// TIA Portal project "Contadores" (V16)

(* hardware
DEVICE "S7-1200 station_1"  S7-1200 Station
   slot 0: "Rack_0"  S7-1200 Rack  Rack  V1.0
   slot 1: "PLC_1"  CPU 1214C AC/DC/Rly  6ES7 214-1BG40-0XB0  V4.4
*)

// ===== PLC "PLC_1"  CPU 1214C AC/DC/Rly =====

VAR_GLOBAL   // PLC tag table "Tabla de variables estándar"
   "Flancos" AT %I0.0 : Bool;
   "Reset" AT %I0.1 : Bool;
   "Contador" AT %MW100 : Int;
   "Relé" AT %Q0.0 : Bool;
   "FlancosDesc" AT %I0.2 : Bool;
   "ResetDesc" AT %I0.3 : Bool;
   "ContadorDesc" AT %MW101 : Int;
   "INT ASC" AT %I0.4 : Bool;
   "INT DESC" AT %I0.5 : Bool;
   "RESET TO 0" AT %I0.6 : Bool;
   "RESET TO 10" AT %I0.7 : Bool;
   "OUT CTU" AT %Q0.1 : Bool;
   "OUT CTD" AT %Q0.2 : Bool;
   "MEMORIA" AT %MD100 : DWord;
END_VAR

// folder: System blocks/Program resources

DATA_BLOCK "IEC_Counter_0_DB"   // DB1
{ S7_Optimized_Access := 'TRUE' }
AUTHOR : Simatic
FAMILY : IEC
NAME : CNTR
VERSION : 1.0
// stored: InstanceOfName IEC_COUNTER
"IEC_COUNTER"
BEGIN
END_DATA_BLOCK

DATA_BLOCK "IEC_Counter_0_DB_1"   // DB2
{ S7_Optimized_Access := 'TRUE' }
AUTHOR : Simatic
FAMILY : IEC
NAME : CNTR
VERSION : 1.0
// stored: InstanceOfName IEC_COUNTER
"IEC_COUNTER"
BEGIN
END_DATA_BLOCK

DATA_BLOCK "IEC_Counter_0_DB_2"   // DB3
{ S7_Optimized_Access := 'TRUE' }
AUTHOR : Simatic
FAMILY : IEC
NAME : CNTR
VERSION : 1.0
// stored: InstanceOfName IEC_COUNTER
"IEC_COUNTER"
BEGIN
END_DATA_BLOCK

// folder: (top level)

ORGANIZATION_BLOCK "Main"   // OB1, LAD, ProgramCycle
TITLE = "Main Program Sweep (Cycle)"
{ S7_Optimized_Access := 'TRUE' }
VERSION : 0.1
   VAR_INPUT
      Initial_Call : Bool;   // Initial call of this OB
      Remanence : Bool;   // =True, if remanent data are available
   END_VAR
BEGIN

REGION Network 1
   // Contador de flanco ascendente CTU
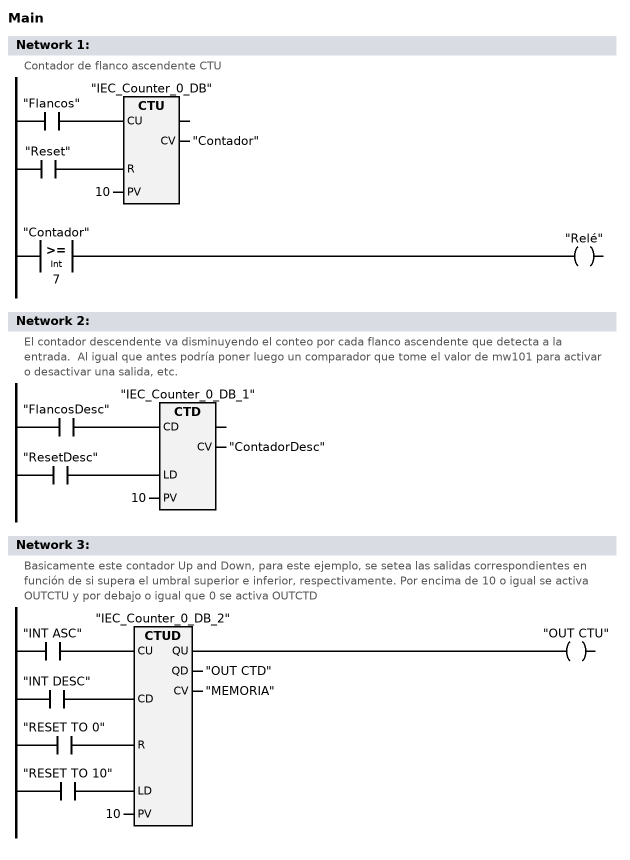
   "IEC_Counter_0_DB".CTU(CU := "Flancos", R := "Reset", PV := 10, CV => "Contador");
   "Relé" := "Contador" >= 7;
END_REGION

REGION Network 2
   // El contador descendente va disminuyendo el conteo por cada flanco ascendente que detecta a la entrada.  Al igual que antes podría poner luego un comparador que tome el valor de mw101 para activar o desactivar una salida, etc.
   "IEC_Counter_0_DB_1".CTD(CD := "FlancosDesc", LD := "ResetDesc", PV := 10, CV => "ContadorDesc");
END_REGION

REGION Network 3
   // Basicamente este contador Up and Down, para este ejemplo, se setea las salidas correspondientes en función de si supera el umbral superior e inferior, respectivamente. Por encima de 10 o igual se activa OUTCTU y por debajo o igual que 0 se activa OUTCTD
   "IEC_Counter_0_DB_2".CTUD(CU := "INT ASC",
                           CD := "INT DESC",
                           R := "RESET TO 0",
                           LD := "RESET TO 10",
                           PV := 10,
                           QD => "OUT CTD",
                           CV => "MEMORIA");
   "OUT CTU" := "IEC_Counter_0_DB_2".QU;
END_REGION
END_ORGANIZATION_BLOCK